Yaskawa INFORM job: COMARC_TEST_ZAKLADKA_4MM.JBI

/JOB
//NAME COMARC_TEST_ZAKLADKA_4MM
//POS
///NPOS 4,4,0,0,0,0
///TOOL 0
///POSTYPE ROBOT
///RECTAN
///RCONF 1,0,0,0,0,0,0,0,0,0,0,0,0,0,0,0,0,0,0,0,0,0,0,0
C00000=535.056,-126.303,-974.722,0.0150,45.0035,0.0266
C00001=558.402,121.549,-978.507,0.0153,45.0047,0.0252
C00002=581.154,69.492,-952.368,-20.5767,34.9799,21.0084
C00003=540.358,121.544,-989.067,0.0152,45.0022,0.0248
///RCONF 0,0,0,0,0,0,0,0,0,0,0,0,0,0,0,0,0,0,0,0,0,0,0,0
BC00000=3071.266
BC00001=3071.266
BC00002=3036.073
BC00003=3071.266
//INST
///DATE 2024/10/23 14:52
///ATTR SC,RW,RJ
////FRAME ROBOT
///GROUP1 RB1,BS1
NOP
REFP 1 C00000 BC00000
REFP 2 C00001 BC00001
MACRO1 MJ#(0) ARGF51
MOVL C00002 BC00002 V=16.7 PL=0
ARCON
COMARCON AMP=2.0 FREQ=2.0 ANGL=45.0 U/D=4800 L/R=0.0 PC=493
MOVL C00003 BC00003 V=6.7
ARCOF
COMARCOF
END
